TYPE ST_Klima_Aussen :
STRUCT
	Temperatur			: REAL;
	Luftfeuchte_rel		: REAL;
	Windgeschwindigkeit	: REAL;
	Regen				: BOOL;
END_STRUCT
END_TYPE

(* stored: Version 1.1.0.1, ProductVersion 3.1.4024.9
   DUT ST_Klima_Aussen: Id {515e9a58-f0af-469f-9801-4ad8d5fd518f} *)
